TYPE ST_Timer :
STRUCT
	
END_STRUCT
END_TYPE

(* stored: Version 1.1.0.1, ProductVersion 3.1.4024.12
   DUT ST_Timer: Id {9d3dd1f9-2f86-4860-b182-f0a7d62ba381} *)
